FUNCTION_BLOCK TESTPAR_COMP (* Test Java emitting of parameters in composite FB type *)
  (* Standard: 61499-2 *)
  (* Version 0.0, 2004-12-15, JHC, Rockwell Automation *)
  (* Compiler header: package fb.rt.test; import fb.rt.math.*; *)
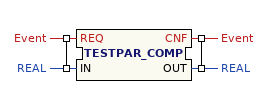
  EVENT_INPUT
    REQ WITH IN; (* Normal Execution Request *)
  END_EVENT
  EVENT_OUTPUT
    CNF WITH OUT; (* Execution Confirmation *)
  END_EVENT
  VAR_INPUT
    IN : REAL;
  END_VAR
  VAR_OUTPUT
    OUT : REAL; (* IN+2.0 *)
  END_VAR
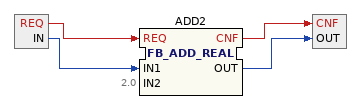
  FBS
    ADD2 : FB_ADD_REAL(IN2 := 2.0);
  END_FBS
  EVENT_CONNECTIONS
    REQ TO ADD2.REQ;
    ADD2.CNF TO CNF;
  END_CONNECTIONS
  DATA_CONNECTIONS
    ADD2.OUT TO OUT;
    IN TO ADD2.IN1;
  END_CONNECTIONS
END_FUNCTION_BLOCK
